// TIA Portal project "scl ejercicio 2" (V11)

(* hardware
DEVICE "S7300/ET200 station_1"  SIMATIC 300-Station
   slot 0: "Perfil soporte_0"  Rail  6ES7 390-1***0-0AA0
   slot 2: "PLC_1"  CPU 313C-2 DP  6ES7 313-6CF03-0AB0  V2.6
      slot 0: "Interfaz MPI_1"  MPI
      slot 1: "Interfaz DP_1"  DP
      slot 2: "DI16/DO16_1"  DI16/DO16
      slot 4: "Contaje_1"  Counter
*)

// ===== PLC "PLC_1"  CPU 313C-2 DP =====

VAR_GLOBAL   // PLC tag table "Tabla de variables estándar"
   "Tag_1" AT %E0.0 : Bool;
   "Tag_2" AT %E0.1 : Bool;
   "Tag_3" AT %E0.2 : Bool;
   "Tag_4" AT %E0.3 : Bool;
   "Tag_5" AT %A0.0 : Bool;
   "Tag_6" AT %A0.1 : Bool;
   "Tag_7" AT %A0.2 : Bool;
   "Tag_8" AT %A0.3 : Bool;
   "Tag_9" AT %T0 : Timer;
   "Tag_10" AT %E0.4 : Bool;
END_VAR

DATA_BLOCK "GRUA AUTOMATICA_DB"   // DB1
{ S7_Optimized_Access := 'FALSE' }
VERSION : 0.1
// stored: InstanceOfName GRUA AUTOMATICA
"GRUA AUTOMATICA"
BEGIN
END_DATA_BLOCK

FUNCTION_BLOCK "GRUA AUTOMATICA"   // FB1, SCL
{ S7_Optimized_Access := 'FALSE' }
VERSION : 0.1
   VAR_INPUT
      MARCHA : Bool;
      FCS2 : Bool;
      FCS3 : Bool;
      FCS4 : Bool;
      FCS5 : Bool;
   END_VAR
   VAR_OUTPUT
      "M1 SUBIR" : Bool;
      "M1 BAJAR" : Bool;
      "M2 DERECHA" : Bool;
      "M2 IZQUIERDA" : Bool;
   END_VAR
   VAR
      M0 : Bool;
      T0 : Bool;
      VISUALIZAR : Time;
   END_VAR
BEGIN
    (* PRIMER CICLO *)
   IF #MARCHA AND #FCS2 AND  #FCS4 THEN  (* SUBIDA HASTA FCS3 *)
     #"M1 BAJAR" := FALSE ;
     #"M1 SUBIR" := TRUE ;
     END_IF;
   IF #"M1 SUBIR" AND #FCS4 AND #FCS3 THEN (* DESPLAZAMIENTO HACIA LA DERECHA HASTA FCS5 *)
     #"M1 SUBIR" := FALSE ;
     #"M2 IZQUIERDA" := FALSE ;
     #"M2 DERECHA" := TRUE ;
     END_IF;

   IF #"M2 DERECHA" AND  #FCS3 AND #FCS5 THEN (* BAJADA HASTA FCS2 *)
     #"M2 DERECHA" := FALSE ;
     #"M1 SUBIR" := FALSE ;
     #"M1 BAJAR" := TRUE ;
   END_IF ;

   IF #FCS5 AND #FCS2  THEN  (* PARO DE BAJADA Y ACTIVACION M0 ALIMENTACION T0 *)
     #"M1 BAJAR" := FALSE ;
     #M0 := TRUE ;
   END_IF;

   "IEC_Timer_0_DB".TON(IN:=#M0, (* TEMPORIZADO CAMBIO DE CICLO 4S *)
                        PT:=T#4S,
                        Q=>#T0,
                        ET=>#VISUALIZAR);

   (* SEGUNDO CICLO *)
   IF #T0 THEN  (* SUBIDA HASTA FCS3 *)
     #M0 := FALSE ;
     #"M1 BAJAR" := FALSE ;
     #"M1 SUBIR" := TRUE ;
   END_IF ;

   IF #"M1 SUBIR" AND #FCS3 AND #FCS5 THEN (*DESPLAZAMIENTO HACIA LA IZQUIERDA HASTA FCS4 *)
     #"M1 SUBIR" := FALSE ;
     #"M2 DERECHA" := FALSE ;
     #"M2 IZQUIERDA" := TRUE ;
   END_IF ;

   IF #"M2 IZQUIERDA" AND #FCS3 AND #FCS4 THEN (* BAJADA HASTA FCS2 *)
     #"M2 IZQUIERDA" := FALSE ;
     #"M1 SUBIR" := FALSE ;
     #"M1 BAJAR" := TRUE ;
   END_IF ;

   IF #"M1 BAJAR" AND #FCS4 AND #FCS2 THEN (* PARO BAJADA FIN SEGUNDO CICLO *)
     #"M1 BAJAR" := FALSE ;
     END_IF;
END_FUNCTION_BLOCK

ORGANIZATION_BLOCK "Main"   // OB1, LAD
TITLE = "Main Program Sweep (Cycle)"
{ S7_Optimized_Access := 'FALSE' }
VERSION : 0.1
   VAR_TEMP
      OB1_EV_CLASS : Byte;   // Bits 0-3 = 1 (Coming event), Bits 4-7 = 1 (Event class 1)
      OB1_SCAN_1 : Byte;   // 1 (Cold restart scan 1 of OB 1), 3 (Scan 2-n of OB 1)
      OB1_PRIORITY : Byte;   // Priority of OB Execution
      OB1_OB_NUMBR : Byte;   // 1 (Organization block 1, OB1)
      OB1_RESERVED_1 : Byte;   // Reserved for system
      OB1_RESERVED_2 : Byte;   // Reserved for system
      OB1_PREV_CYCLE : Int;   // Cycle time of previous OB1 scan (milliseconds)
      OB1_MIN_CYCLE : Int;   // Minimum cycle time of OB1 (milliseconds)
      OB1_MAX_CYCLE : Int;   // Maximum cycle time of OB1 (milliseconds)
      OB1_DATE_TIME : Date_And_Time;   // Date and time OB1 started
   END_VAR
BEGIN

REGION Network 1
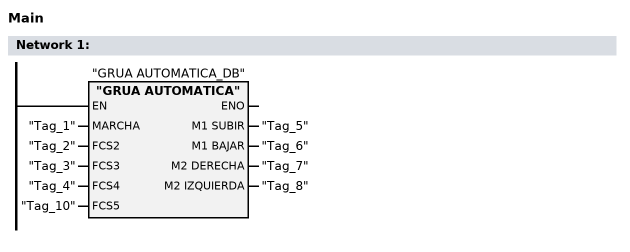
   RUNG wire#powerrail
      "GRUA AUTOMATICA_DB"(MARCHA := "Tag_1", FCS2 := "Tag_2", FCS3 := "Tag_3", FCS4 := "Tag_4", FCS5 := "Tag_10", "M1 SUBIR" => "Tag_5", "M1 BAJAR" => "Tag_6", "M2 DERECHA" => "Tag_7", "M2 IZQUIERDA" => "Tag_8")
   END_RUNG
   // the same network as SCL:
   "GRUA AUTOMATICA_DB"(MARCHA := "Tag_1",   // "GRUA AUTOMATICA"
                        FCS2 := "Tag_2",
                        FCS3 := "Tag_3",
                        FCS4 := "Tag_4",
                        FCS5 := "Tag_10",
                        "M1 SUBIR" => "Tag_5",
                        "M1 BAJAR" => "Tag_6",
                        "M2 DERECHA" => "Tag_7",
                        "M2 IZQUIERDA" => "Tag_8");
END_REGION
END_ORGANIZATION_BLOCK